FUNCTION_BLOCK FB_Clock
VAR_INPUT
	bStart : BOOL;
	bStop : BOOL;
	fCycleTime : REAL;
END_VAR
VAR_OUTPUT
	fTimeInSeconds : REAL;
END_VAR
VAR
END_VAR



IF bStart = TRUE AND bStop = FALSE THEN
	fTimeInSeconds := fTimeInSeconds + fCycleTime;
ELSE
	fTimeInSeconds := 0.0;
END_IF

END_FUNCTION_BLOCK

(* stored: Version 1.1.0.1, ProductVersion 3.1.4024.10
   POU FB_Clock: Id {cd260362-2b58-4b71-929f-8a02100da9e0}, SpecialFunc None *)
